// TwinCAT 3 PLC project Strategy_Pattern
// ProgramVersion: 3.1.4024.0
// libraries:
//   Tc2_Standard, * (Beckhoff Automation GmbH)
//   Tc2_System, * (Beckhoff Automation GmbH)
//   Tc3_Module, * (Beckhoff Automation GmbH)
// project tree:
//   Classes/ SomeCyclicClass.TcPOU
//   Loggers/ CSVWriter.TcPOU, ITF_Writer.TcIO, JsonWriter.TcPOU, TextWriter.TcPOU
//   / PlcTask.TcTTO
//   POUs/ MAIN.TcPOU
// (motion and I/O tree: see PLC project simple_factory_pattern)
// real-time tasks:
//   TASK PlcTask: cycle T#10ms, priority 20, ADS port 350
//   TASK PlcTask1: cycle T#10ms, priority 21, ADS port 351
//   TASK PlcTask2: cycle T#10ms, priority 22, ADS port 352
//   TASK PlcTask3: cycle T#10ms, priority 23, ADS port 353

CONFIGURATION Strategy_Pattern
    RESOURCE PLC ON TwinCAT3
        TASK PlcTask(INTERVAL := T#10ms, PRIORITY := 23);
        PROGRAM MAIN WITH PlcTask : MAIN;
    END_RESOURCE
END_CONFIGURATION

// ---- Loggers/ITF_Writer.TcIO
INTERFACE ITF_Writer

METHOD WriteMessage : BOOL
VAR_INPUT
	SomeString : STRING(80);
END_VAR
END_METHOD

END_INTERFACE

// ---- POUs/MAIN.TcPOU
PROGRAM MAIN
VAR
	myCsvWriter : CSVWriter;
	myJsonWriter : JsonWriter;
	myTextWriter : TextWriter;
	myObject : SomeCyclicClass := (MyWriter := myTextWriter);
	runOperation1: BOOL;
	runOperation2: BOOL;
	runOperation3: BOOL;
	xtest: BOOL;
END_VAR

IF runOperation1 THEN
	runOperation1 := FALSE;
	myObject.MyWriter := myJsonWriter;
	myObject.DoSomething();
END_IF

IF runOperation2 THEN
	runOperation2 := FALSE;
	myObject.MyWriter := myTextWriter;
	myObject.DoSomething();
END_IF

IF runOperation3 THEN
	runOperation3 := FALSE;
	myObject.MyWriter := myCsvWriter;
	myObject.DoSomething();
END_IF

IF xtest THEN
	xtest := FALSE;
	myObject.MyWriter := myCsvWriter;
END_IF

END_PROGRAM

// ---- Loggers/CSVWriter.TcPOU
FUNCTION_BLOCK CSVWriter IMPLEMENTS ITF_Writer
VAR
END_VAR

METHOD WriteMessage : BOOL
VAR_INPUT
	SomeString	: STRING(80);
END_VAR
ADSLOGSTR(msgCtrlMask := ADSLOG_MSGTYPE_LOG, msgFmtStr := 'I wrote a CSV line with: %s',strArg := SomeString);
END_METHOD

END_FUNCTION_BLOCK

// ---- Loggers/JsonWriter.TcPOU
FUNCTION_BLOCK JsonWriter IMPLEMENTS ITF_Writer
VAR
END_VAR

METHOD WriteMessage : BOOL
VAR_INPUT
	SomeString	: STRING(80);
END_VAR
ADSLOGSTR(msgCtrlMask := ADSLOG_MSGTYPE_LOG, msgFmtStr := 'I wrote a JSON line with: %s',strArg := SomeString);
END_METHOD

END_FUNCTION_BLOCK

// ---- Loggers/TextWriter.TcPOU
FUNCTION_BLOCK TextWriter IMPLEMENTS ITF_Writer
VAR
END_VAR

METHOD WriteMessage : BOOL
VAR_INPUT
	SomeString	: STRING(80);
END_VAR
ADSLOGSTR(msgCtrlMask := ADSLOG_MSGTYPE_LOG, msgFmtStr := 'I wrote a Text line with: %s',strArg := SomeString);
END_METHOD

END_FUNCTION_BLOCK

// ---- Classes/SomeCyclicClass.TcPOU
FUNCTION_BLOCK SomeCyclicClass
VAR
	_myWriter : ITF_Writer;
END_VAR

METHOD DoSomething : BOOL
VAR_INPUT
END_VAR
///////Perform some operations////////

IF _myWriter <> 0 THEN
	_myWriter.WriteMessage('I did a job :-)');
END_IF
END_METHOD

PROPERTY MyWriter : ITF_Writer
GET
MyWriter := _myWriter;
END_GET
SET
_myWriter := MyWriter;
END_SET
END_PROPERTY

END_FUNCTION_BLOCK
